INTERFACE ITcoToggleTask EXTENDS ITcoObject

(*~
	<docu>
		<summary>
			Use to set the state of the '''TcoToggleTask''' to the value '''FALSE'''.
		</summary>
	</docu>
~*)
METHOD Off : BOOL
END_METHOD

(*~
	<docu>
		<summary>
			Use to set the state of the '''TcoToggleTask''' to the value '''TRUE'''.
		</summary>
	</docu>
~*)
METHOD On : BOOL
END_METHOD

(*~
	<docu>
		<summary>
			Use to toggle the state of the '''TcoToggleTask'''.
		</summary>
	</docu>
~*)
METHOD Toggle : BOOL
END_METHOD

END_INTERFACE

(* stored: Version 1.1.0.1
   Itf ITcoToggleTask: Id {01c40efa-562e-0078-1855-26cbab73f0bb}
   Method Off: Id {2e350264-5024-0bd9-0fd7-5fd987d34952}
   Method On: Id {c6a7c9ba-3e57-01fa-1c81-6d07c4c3c9f2}
   Method Toggle: Id {e4190899-2a97-08fb-33a3-b2ea419c86b2} *)
